FUNCTION_BLOCK SocketSendTask IMPLEMENTS ITask
VAR_INPUT
END_VAR
VAR_OUTPUT
END_VAR
VAR
	iState: INT;
	_done: BOOL;
	_busy: BOOL;
	_error: BOOL;
	_execute : BOOL;
	fbSocketSend : Tc2_TcpIp.FB_SocketSend;
END_VAR

CASE iState OF
	0:
		IF _execute THEN
			_done := FALSE;
			_busy := TRUE;
			_error := FALSE;
			fbSocketSend.bExecute := TRUE;
			IF fbSocketSend.bBusy THEN
				iState := 10;
				_execute := false;
			END_IF
		END_IF
	10:
		IF NOT fbSocketSend.bBusy THEN
			IF NOT fbSocketSend.bError THEN
				_done := TRUE;
			ELSE
				_error := TRUE;
			END_IF
			_busy := FALSE;
			fbSocketSend.bExecute := FALSE;
			iState := 0;
		END_IF
END_CASE

fbSocketSend(tTimeout := Tc2_System.DEFAULT_ADS_TIMEOUT);

METHOD Abort : BOOL
fbSocketSend.bExecute := FALSE;
_busy := FALSE;
_execute := FALSE;
Abort := TRUE;
iState := 0;
END_METHOD

PROPERTY Busy : BOOL
GET
Busy := _busy;
END_GET
END_PROPERTY

PROPERTY Done : BOOL
GET
Done := _done;
END_GET
END_PROPERTY

PROPERTY Error : BOOL
GET
Error := _error;
END_GET
END_PROPERTY

METHOD Execute : BOOL
VAR_INPUT
	DataToSend : POINTER TO BYTE;
	DataLength : UDINT;
END_VAR
IF NOT fbSocketSend.bBusy THEN
	fbSocketSend.pSrc := DataToSend;
	fbSocketSend.cbLen := DataLength;
	Execute := _execute := true;
END_IF
END_METHOD

PROPERTY PUBLIC RemoteSocket : T_HSOCKET
GET // PUBLIC
RemoteSocket := fbSocketSend.hSocket;
END_GET
SET // PUBLIC
fbSocketSend.hSocket := RemoteSocket;
END_SET
END_PROPERTY

END_FUNCTION_BLOCK

(* stored: Version 1.1.0.1, ProductVersion 3.1.4024.12
   POU SocketSendTask: Id {4f030919-0a98-4351-809a-94c4dc20c30b}, SpecialFunc None
   Method Abort: Id {e0715338-7996-4356-a55e-29c43a6231d4}
   Property Busy: Id {a6ad668d-5d57-4e2c-9179-e8b3b99d79df}
   Get Get: Id {5fc82b9b-c42a-4a3f-98c0-ff24bdbf3ac5}
   Property Done: Id {84c25007-6a09-4d8f-b82a-218e94d68125}
   Get Get: Id {31fa1c99-2564-4453-b380-e92595d80254}
   Property Error: Id {fbe17f00-50f6-488a-b5d5-2280f458be8e}
   Get Get: Id {cf7c4b69-35a1-443a-8485-9866aa03d9cf}
   Method Execute: Id {f48cef18-e120-4f1a-be71-36cbb216941d}
   Property RemoteSocket: Id {05fdfbd5-8764-4c89-b7bf-7538d3011211}
   Get Get: Id {1c47167f-0203-460b-b516-2c1b20440c76}
   Set Set: Id {64cb43d3-5066-4c29-8a83-7e712b3da039} *)
